// Example 3 - StitchedSegments: ONE cam table, the same 18 points as example 2, assembled from pieces.
//
//   Mover 1 = master, runs at constant velocity around the track.
//   Mover 2 = slave, follows Mover 1 through a cam table that covers one full lap (1500 mm).
//
// The clothoid exists once, as a module-relative piece: BuildCurveModule runs FB_XtsBallCamBuilder for ONE curve
// module at the origin (aCurvePoints). The track is a list of segments, and FB_XtsCamStitcher pastes the piece
// wherever the list says "Curve" (action BuildTable). Change the straights = change the list, the clothoid stays.
//
// How to run (online view, with MAIN.eExample = StitchedSegments):  bStart -> watch eState -> bStop.   On Error: bReset.
// Watch fGapActual while it runs (115 on the straights) and fStitchMaxDeviation: the difference to the example 2
// table, expect ~1e-9 mm.
PROGRAM PRG_Example3
VAR CONSTANT
	// --- track geometry (mm) ---
	TRACK_LENGTH			: LREAL := 1500.0;	// = modulo factor of both mover axes
	STRAIGHT_1_START		: LREAL := 0.0;
	CURVE_1_START			: LREAL := 250.0;
	STRAIGHT_2_START		: LREAL := 750.0;
	CURVE_2_START			: LREAL := 1000.0;
	MODULE_LENGTH			: LREAL := 500.0;	// one 180 deg curve module (AT2050)

	// --- the ball clamped between the two movers (see example 2) ---
	BALL_DISTANCE			: LREAL := 115.0;	// mm between the two jaws, measured along the ball's path
	BALL_OFFSET				: LREAL := 103.03;	// mm the ball (and the jaws) sit outboard of the mover path
	TABLE_START				: LREAL := 180.0;	// master position of the first table point. Any point on straight 1
												// that keeps every ramp clear of the 1500 -> 0 wrap works (103 < x < 266).

	// --- the clothoid as ONE module-relative piece ---
	CURVE_TABLE_LENGTH		: LREAL := 620.0;	// mm of master one curve piece covers, measured from the module start.
												// Must reach past the builder's last exit knot (603): the trailing ball
												// keeps the cam busy 103 mm after the module ends. The builder errors if not.
	MAX_CURVE_POINTS		: UDINT := 16;

	// --- demo dynamics ---
	MASTER_VELOCITY			: LREAL := 300.0;	// mm/s, Mover 1 while running
	POSITIONING_VELOCITY	: LREAL := 200.0;	// mm/s, Mover 2 while pre-positioning

	CAM_TABLE_ID			: MC_CAM_ID := 1;	// NC > Tables > Table 1 (Ex 1-4) > Mover 2
	MAX_CAM_POINTS			: UDINT := 32;		// 8 per curve + 2 = 18, the rest is room for more segments
	PLC_ERROR_ID			: UDINT := 16#FFFF_FFFF;	// not an NC error: builder or stitcher refused, see sTableError
END_VAR
VAR
	// --- commands: set TRUE in the online view, they reset themselves ---
	bStart				: BOOL;
	bStop				: BOOL;
	bReset				: BOOL;
	eState				: E_State;

	// --- cam table data: nCamPoints points, loaded into NC table CAM_TABLE_ID ---
	aCamPoints			: ARRAY[1..MAX_CAM_POINTS] OF MC_MotionFunctionPoint;
	nCamPoints			: UDINT;		// points actually used (18)
	stCamTable			: MC_CAM_REF;

	// --- the clothoid piece and the stitcher ---
	fbBuilder			: FB_XtsBallCamBuilder;	// computes the clothoid points of one module
	aCurvePoints		: ARRAY[1..MAX_CURVE_POINTS] OF MC_MotionFunctionPoint;	// 10 points, master 0..CURVE_TABLE_LENGTH from the module start
	nCurvePoints		: UDINT;
	fbStitcher			: FB_XtsCamStitcher;	// layout + curve piece -> one lap table
	aCheckPoints		: ARRAY[1..MAX_CAM_POINTS] OF MC_MotionFunctionPoint;	// the example 2 table, built next to it for comparison
	fStitchMaxDeviation	: LREAL;		// largest difference to the example 2 table in mm (expect ~1e-9, -1 = no comparison)

	// --- function blocks ---
	fbPowerMover1		: MC_Power;
	fbPowerMover2		: MC_Power;
	fbResetMover1		: MC_Reset;
	fbResetMover2		: MC_Reset;
	fbCamTableSelect	: MC_CamTableSelect;			// PLC array -> NC cam table
	fbReadTable			: MC_ReadCamTableSlaveDynamics;	// "where does the table want the slave for this master position?"
	fbMoveRelMover2		: MC_MoveRelative;
	fbCamIn				: MC_CamIn;
	fbMoveVeloMover1	: MC_MoveVelocity;
	fbHaltMover1		: MC_Halt;
	fbCamOut			: MC_CamOut;

	// --- live values worth watching ---
	fMover1Pos			: LREAL;	// modulo set position of Mover 1 (0..1500)
	fMover2Pos			: LREAL;	// modulo set position of Mover 2 (0..1500)
	fGapActual			: LREAL;	// how far Mover 2 is behind Mover 1 right now (along the track)
	fGapWanted			: LREAL;	// what the table asked for at coupling time
	fMasterInTable		: LREAL;	// fMover1Pos mapped into the master range of the table (TABLE_START .. +1500)
	bError				: BOOL;
	nErrorID			: UDINT;
	sTableError			: STRING(255);	// why the PLC side refused: builder or stitcher (nErrorID = PLC_ERROR_ID)

	// --- scratch ---
	i					: UINT;
END_VAR

// update axis status every cycle
GVL_Axes.Mover1();
GVL_Axes.Mover2();

// live gap: Mover 1 position minus Mover 2 position, wrapped to 0..1500
fMover1Pos := GVL_Axes.Mover1.NcToPlc.ModuloSetPos;
fMover2Pos := GVL_Axes.Mover2.NcToPlc.ModuloSetPos;
fGapActual := fMover1Pos - fMover2Pos;
IF fGapActual < 0.0 THEN
	fGapActual := fGapActual + TRACK_LENGTH;
END_IF

CASE eState OF
	E_State.Idle:
		IF bStart THEN
			bStart := FALSE;
			eState := E_State.Enable;
		END_IF

	E_State.Enable:
		fbPowerMover1.Enable := TRUE;
		fbPowerMover1.Enable_Positive := TRUE;
		fbPowerMover1.Enable_Negative := TRUE;
		fbPowerMover2.Enable := TRUE;
		fbPowerMover2.Enable_Positive := TRUE;
		fbPowerMover2.Enable_Negative := TRUE;
		IF fbPowerMover1.Status AND fbPowerMover2.Status THEN
			eState := E_State.Decouple;
		END_IF

	E_State.Decouple:
		// An earlier run may have left Mover 2 coupled: the NC keeps the coupling through an axis error and MC_Reset
		// does not clear it. MC_CamTableSelect refuses to overwrite a table that a coupled axis is using (0x4A26).
		IF NOT fbCamOut.Execute THEN
			IF GVL_Axes.Mover2.Status.Coupled THEN
				fbCamOut.Execute := TRUE;
			ELSE
				eState := E_State.BuildTable;
			END_IF
		ELSIF fbCamOut.Done THEN
			fbCamOut.Execute := FALSE;
			eState := E_State.BuildTable;
		END_IF

	E_State.BuildTable:
		// fill the point array once, then hand it to the NC (overwrites cam table CAM_TABLE_ID)
		IF NOT fbCamTableSelect.Execute THEN
			BuildTable();
		END_IF
		IF nCamPoints > 0 THEN		// = 0: builder or stitcher refused, the error check below picks up sTableError
			fbCamTableSelect.Periodic := TRUE;		// one table = one lap, repeat forever
			fbCamTableSelect.CamTableID := CAM_TABLE_ID;
			fbCamTableSelect.Execute := TRUE;
			IF fbCamTableSelect.Done THEN
				fbCamTableSelect.Execute := FALSE;
				eState := E_State.ReadTable;
			END_IF
		END_IF

	E_State.ReadTable:
		// Mover 1 stays where it is. Ask the NC what slave position the table wants for it.
		// The table master runs from TABLE_START to TABLE_START + 1500, so a track position
		// below the table start is one lap further on in the table.
		IF NOT fbReadTable.Execute THEN
			fMasterInTable := fMover1Pos;
			IF fMasterInTable < TABLE_START THEN
				fMasterInTable := fMasterInTable + TRACK_LENGTH;
			END_IF
			fbReadTable.CamTableID := CAM_TABLE_ID;
			fbReadTable.MasterPosition := fMasterInTable;
		END_IF
		fbReadTable.Execute := TRUE;
		IF fbReadTable.Done THEN
			fbReadTable.Execute := FALSE;
			// table: slave = master - gap   ->   gap = master - slave
			fGapWanted := fMasterInTable - fbReadTable.SlavePosition;
			// Mover 1 stands still, so this relative move can never run into it:
			// positive = Mover 2 closes up from behind, negative = Mover 2 backs off a little
			fbMoveRelMover2.Distance := fGapActual - fGapWanted;
			eState := E_State.Preposition;
		END_IF

	E_State.Preposition:
		fbMoveRelMover2.Velocity := POSITIONING_VELOCITY;
		fbMoveRelMover2.Execute := TRUE;
		IF fbMoveRelMover2.Done THEN
			fbMoveRelMover2.Execute := FALSE;
			eState := E_State.CamIn;
		END_IF

	E_State.CamIn:
		fbCamIn.CamTableID := CAM_TABLE_ID;
		fbCamIn.StartMode := MC_STARTMODE_ABSOLUTE;		// table master axis = Mover 1 track position
		fbCamIn.MasterOffset := 0.0;
		fbCamIn.SlaveOffset := 0.0;
		fbCamIn.MasterScaling := 1.0;
		fbCamIn.SlaveScaling := 1.0;
		// let the NC pick the slave offset so Mover 2 never jumps at coupling.
		// After the pre-positioning above that offset is 0 (or whole laps), so the table gaps apply 1:1.
		fbCamIn.Options.SlaveScalingMode := MC_CAMSCALING_AUTOOFFSET;
		fbCamIn.Execute := TRUE;
		IF fbCamIn.InSync THEN
			fbCamIn.Execute := FALSE;
			eState := E_State.Run;
		END_IF

	E_State.Run:
		// only the master is commanded - the slave is driven by the cam
		fbMoveVeloMover1.Velocity := MASTER_VELOCITY;
		fbMoveVeloMover1.Direction := MC_Positive_Direction;
		fbMoveVeloMover1.Execute := TRUE;
		IF bStop THEN
			bStop := FALSE;
			fbMoveVeloMover1.Execute := FALSE;
			eState := E_State.Stopping;
		END_IF

	E_State.Stopping:
		fbHaltMover1.Execute := TRUE;
		IF fbHaltMover1.Done THEN
			fbHaltMover1.Execute := FALSE;
			eState := E_State.CamOut;
		END_IF

	E_State.CamOut:
		fbCamOut.Execute := TRUE;
		IF fbCamOut.Done THEN
			fbCamOut.Execute := FALSE;
			eState := E_State.Idle;
		END_IF

	E_State.Error:
		fbCamTableSelect.Execute := FALSE;
		fbReadTable.Execute := FALSE;
		fbMoveRelMover2.Execute := FALSE;
		fbCamIn.Execute := FALSE;
		fbMoveVeloMover1.Execute := FALSE;
		// a slave error does not stop the master: halt Mover 1 if it is still running and not in error itself
		fbHaltMover1.Execute := NOT GVL_Axes.Mover1.Status.Error AND GVL_Axes.Mover1.Status.Moving;
		fbCamOut.Execute := FALSE;
		IF bReset THEN
			bReset := FALSE;
			fbResetMover1.Execute := TRUE;
			fbResetMover2.Execute := TRUE;
			eState := E_State.Resetting;
		END_IF

	E_State.Resetting:
		IF (fbResetMover1.Done OR fbResetMover1.Error) AND (fbResetMover2.Done OR fbResetMover2.Error) THEN
			fbResetMover1.Execute := FALSE;
			fbResetMover2.Execute := FALSE;
			bError := FALSE;
			nErrorID := 0;
			sTableError := '';
			eState := E_State.Idle;
		END_IF
END_CASE

// any error anywhere -> Error state
IF eState <> E_State.Error AND eState <> E_State.Resetting THEN
	IF GVL_Axes.Mover1.Status.Error THEN
		nErrorID := GVL_Axes.Mover1.Status.ErrorID;
	ELSIF GVL_Axes.Mover2.Status.Error THEN
		nErrorID := GVL_Axes.Mover2.Status.ErrorID;
	ELSIF fbPowerMover1.Error THEN
		nErrorID := fbPowerMover1.ErrorID;
	ELSIF fbPowerMover2.Error THEN
		nErrorID := fbPowerMover2.ErrorID;
	ELSIF sTableError <> '' THEN
		nErrorID := PLC_ERROR_ID;
	ELSIF fbCamTableSelect.Error THEN
		nErrorID := fbCamTableSelect.ErrorID;
	ELSIF fbReadTable.Error THEN
		nErrorID := fbReadTable.ErrorID;
	ELSIF fbMoveRelMover2.Error THEN
		nErrorID := fbMoveRelMover2.ErrorID;
	ELSIF fbCamIn.Error THEN
		nErrorID := fbCamIn.ErrorID;
	ELSIF fbMoveVeloMover1.Error THEN
		nErrorID := fbMoveVeloMover1.ErrorID;
	ELSIF fbHaltMover1.Error THEN
		nErrorID := fbHaltMover1.ErrorID;
	ELSIF fbCamOut.Error THEN
		nErrorID := fbCamOut.ErrorID;
	END_IF
	IF nErrorID <> 0 THEN
		bError := TRUE;
		eState := E_State.Error;
	END_IF
END_IF

// call every function block once per cycle
fbPowerMover1(Axis := GVL_Axes.Mover1);
fbPowerMover2(Axis := GVL_Axes.Mover2);
fbResetMover1(Axis := GVL_Axes.Mover1);
fbResetMover2(Axis := GVL_Axes.Mover2);
fbCamTableSelect(Master := GVL_Axes.Mover1, Slave := GVL_Axes.Mover2, CamTable := stCamTable);
fbReadTable();
fbMoveRelMover2(Axis := GVL_Axes.Mover2);
fbCamIn(Master := GVL_Axes.Mover1, Slave := GVL_Axes.Mover2);
fbMoveVeloMover1(Axis := GVL_Axes.Mover1);
fbHaltMover1(Axis := GVL_Axes.Mover1);
fbCamOut(Slave := GVL_Axes.Mover2);

ACTION BuildCurveModule:
// ONE curve module as a module-relative cam piece: master 0..CURVE_TABLE_LENGTH measured from the module start,
// slave measured from the same origin with the ball gap included (point 1 = (0, -BALL_DISTANCE)). The same geometry
// as example 2, just for a single module at the origin: 8 clothoid points (ramp / plateau / ramp / line at the
// entry, mirrored at the exit) plus one 1:1 point at each end = 10 points.
//
// BuildTable pastes the 8 inner points wherever the layout says "Curve". Tuning the clothoid (the knot defaults
// in FB_XtsBallCamBuilder) happens here, once, independent of where the curves are on the track.
fbBuilder.fMasterStart		:= 0.0;
fbBuilder.fMasterEnd		:= CURVE_TABLE_LENGTH;
fbBuilder.fBallDistance		:= BALL_DISTANCE;
fbBuilder.fBallOffset		:= BALL_OFFSET;
fbBuilder.nCurves			:= 1;
fbBuilder.aCurveStart[1]	:= 0.0;
fbBuilder.fModuleLength		:= MODULE_LENGTH;
// fTransLength, aEntryKnots, aExitKnots keep the FB defaults (tuned for 115 mm / 103 mm on AT2050 modules)
fbBuilder.pPoints			:= ADR(aCurvePoints);
fbBuilder.nMaxPoints		:= MAX_CURVE_POINTS;

IF fbBuilder.Build() THEN
	nCurvePoints := fbBuilder.nPoints;		// 10
ELSE
	nCurvePoints := 0;
	sTableError := fbBuilder.sError;
END_IF
END_ACTION

ACTION BuildTable:
// The same table as example 2 (18 points, master TABLE_START .. +1500), assembled differently:
// the clothoid exists once, as a module-relative piece (BuildCurveModule -> aCurvePoints), and the track is a list
// of segments. FB_XtsCamStitcher walks the list, pastes the 8 inner curve points at every "Curve" (shifted by the
// running master position) and lets the straights run 1:1 without any points of their own.
// Changing a straight = changing a length in the list. The clothoid piece is untouched.
//
// Rules for the list: start and end on a straight (the table's first/last point must be 1:1), and every straight
// after a curve must be longer than the curve piece overhangs the module (103 mm with the default knots). The
// stitcher reports an error otherwise.
sTableError := '';
nCamPoints := 0;

BuildCurveModule();
IF nCurvePoints = 0 THEN RETURN; END_IF		// sTableError is set

// one lap starting at TABLE_START (180): rest of straight 1 | curve 1 | straight 2 | curve 2 | start of straight 1
fbStitcher.aLayout[1].eKind := E_SegmentKind.Straight;	fbStitcher.aLayout[1].fLength := CURVE_1_START - TABLE_START;			//  70
fbStitcher.aLayout[2].eKind := E_SegmentKind.Curve;		fbStitcher.aLayout[2].fLength := MODULE_LENGTH;							// 500
fbStitcher.aLayout[3].eKind := E_SegmentKind.Straight;	fbStitcher.aLayout[3].fLength := CURVE_2_START - STRAIGHT_2_START;		// 250
fbStitcher.aLayout[4].eKind := E_SegmentKind.Curve;		fbStitcher.aLayout[4].fLength := MODULE_LENGTH;							// 500
fbStitcher.aLayout[5].eKind := E_SegmentKind.Straight;	fbStitcher.aLayout[5].fLength := TABLE_START - STRAIGHT_1_START;		// 180
fbStitcher.nSegments	:= 5;
fbStitcher.fMasterStart	:= TABLE_START;
fbStitcher.fStraightGap	:= BALL_DISTANCE;
fbStitcher.pCurvePoints	:= ADR(aCurvePoints[2]);	// the 8 clothoid points, without the 1:1 end points of the piece
fbStitcher.nCurvePoints	:= nCurvePoints - 2;
fbStitcher.pPoints		:= ADR(aCamPoints);
fbStitcher.nMaxPoints	:= MAX_CAM_POINTS;

IF NOT fbStitcher.Build() THEN
	sTableError := fbStitcher.sError;
	RETURN;
END_IF
IF ABS(fbStitcher.fLength - TRACK_LENGTH) > 0.001 THEN
	sTableError := 'layout does not add up to one lap';
	RETURN;
END_IF
nCamPoints := fbStitcher.nPoints;		// 18

// describe the array to the NC
stCamTable.pArray		:= ADR(aCamPoints);
stCamTable.ArraySize	:= nCamPoints * SIZEOF(MC_MotionFunctionPoint);
stCamTable.TableType	:= MC_TABLETYPE_MOTIONFUNCTION;
stCamTable.NoOfRows		:= nCamPoints;
stCamTable.NoOfColumns	:= 1;

// self-check: build the example 2 table next to it and compare point by point
fbBuilder.fMasterStart		:= TABLE_START;
fbBuilder.fMasterEnd		:= TABLE_START + TRACK_LENGTH;
fbBuilder.nCurves			:= 2;
fbBuilder.aCurveStart[1]	:= CURVE_1_START;
fbBuilder.aCurveStart[2]	:= CURVE_2_START;
fbBuilder.pPoints			:= ADR(aCheckPoints);
fbBuilder.nMaxPoints		:= MAX_CAM_POINTS;
fStitchMaxDeviation := 0.0;
IF fbBuilder.Build() AND_THEN fbBuilder.nPoints = nCamPoints THEN
	FOR i := 1 TO UDINT_TO_UINT(nCamPoints) DO
		fStitchMaxDeviation := MAX(fStitchMaxDeviation, ABS(aCamPoints[i].MasterPos - aCheckPoints[i].MasterPos));
		fStitchMaxDeviation := MAX(fStitchMaxDeviation, ABS(aCamPoints[i].SlavePos  - aCheckPoints[i].SlavePos));
	END_FOR
ELSE
	fStitchMaxDeviation := -1.0;		// could not compare
END_IF
END_ACTION

END_PROGRAM

(* stored: Version 1.1.0.1
   POU PRG_Example3: Id {6af4574e-6aee-4c88-b6a6-7cc3f68f9255}, SpecialFunc None
   Action BuildCurveModule: Id {b3025b6b-af72-4b32-8747-80b8585643d9}
   Action BuildTable: Id {f826822e-8c3d-405b-bc30-b936ed7c0a3f} *)
